(* PLC project SafeLOGIC, BrAutomation SafeDESIGNER  5.24.1.0 *)
(* stored: companyURL http://www.br-automation.com, creationDateTime Fri Nov 28 15:23:45 2025 *)

PROGRAM ERV_Fan

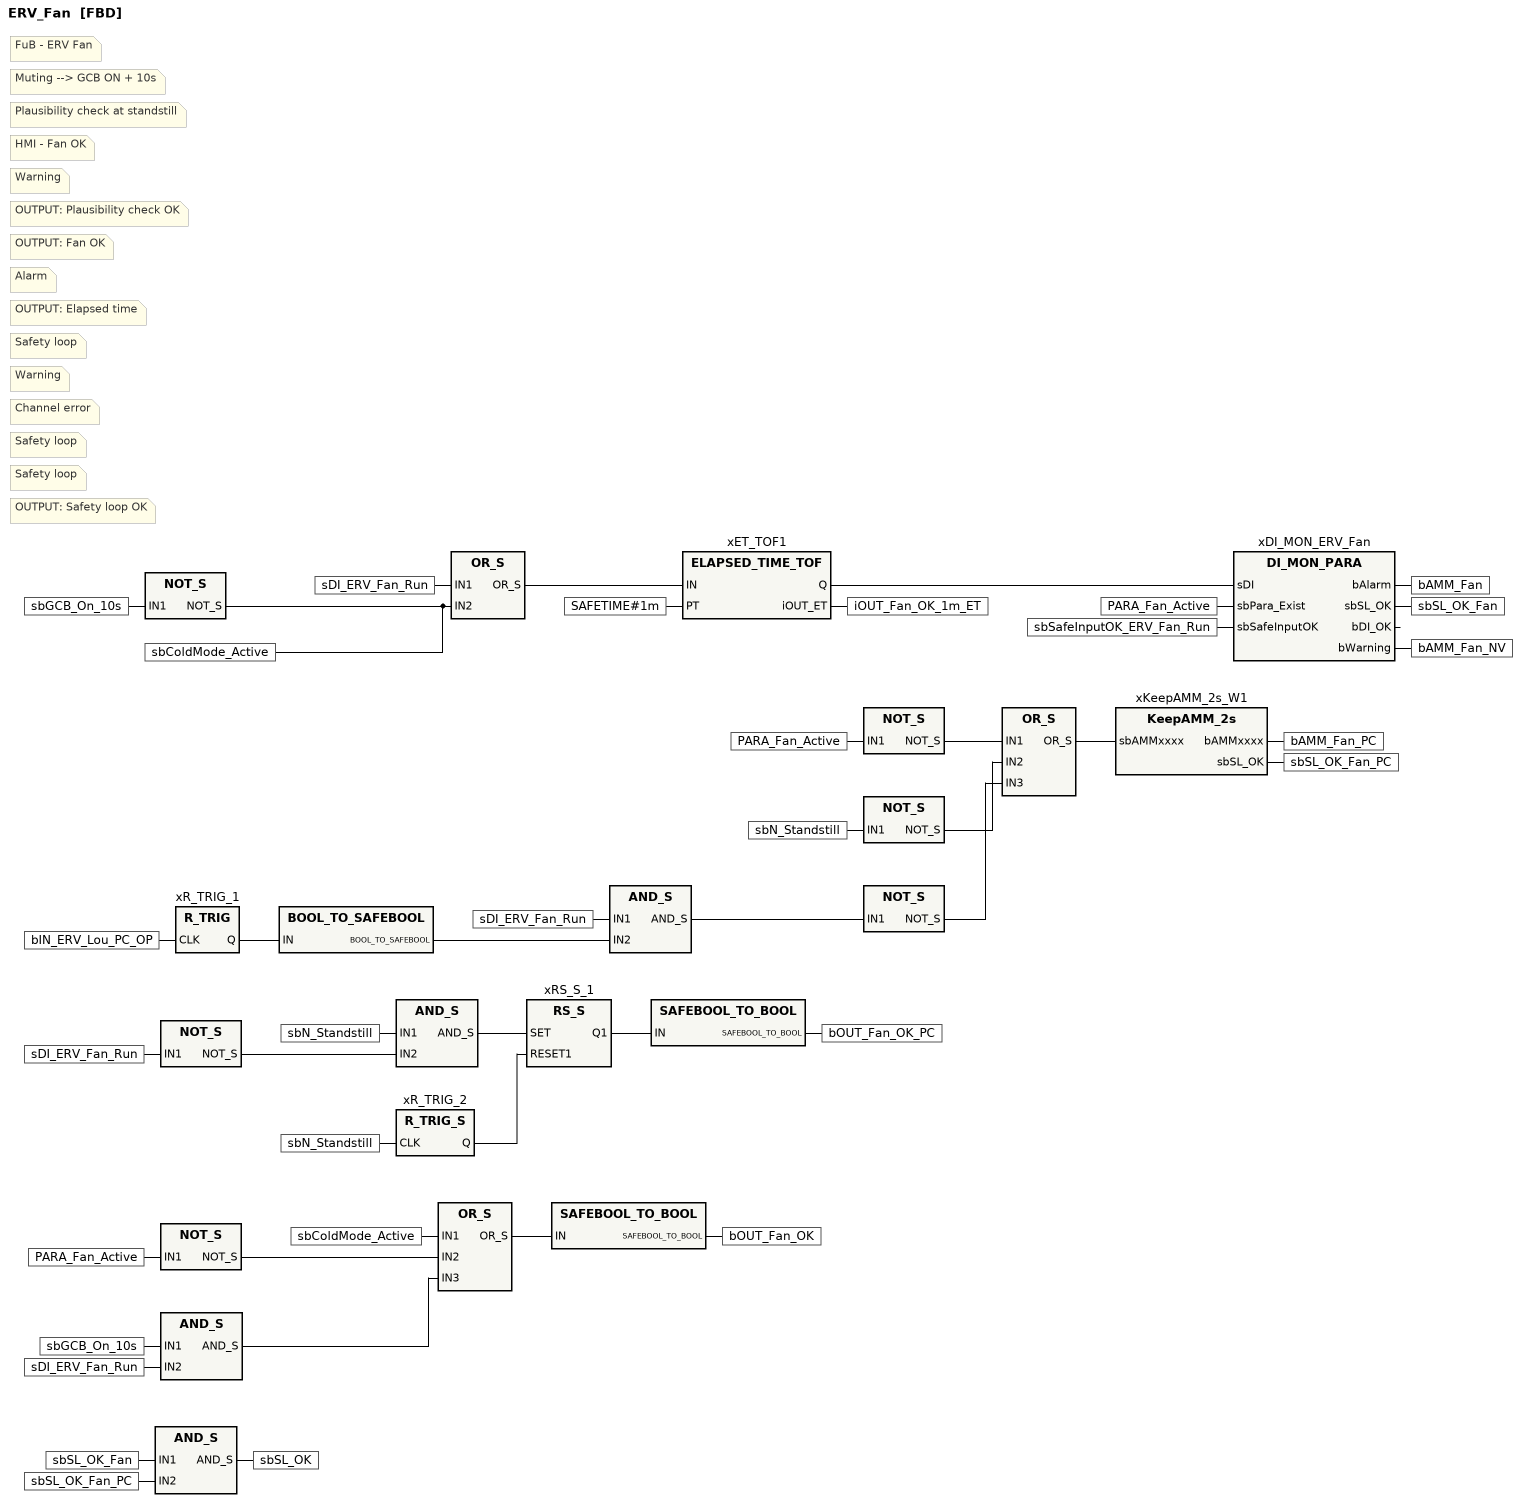
(* FBD diagram, written out as Structured Text *)
(* FuB - ERV Fan *)
(* Alarm *)
(* Safety loop *)
xET_TOF1(IN := OR_S(sDI_ERV_Fan_Run, sbColdMode_Active, NOT_S(sbGCB_On_10s)), PT := SAFETIME#1m);
xDI_MON_ERV_Fan(sDI := xET_TOF1.Q, sbPara_Exist := PARA_Fan_Active, sbSafeInputOK := sbSafeInputOK_ERV_Fan_Run);
bAMM_Fan := xDI_MON_ERV_Fan.bAlarm;
(* Muting --> GCB ON + 10s *)
(* Channel error *)
(* Warning *)
(* OUTPUT: Elapsed time *)
iOUT_Fan_OK_1m_ET := xET_TOF1.iOUT_ET;
bAMM_Fan_NV := xDI_MON_ERV_Fan.bWarning;
sbSL_OK_Fan := xDI_MON_ERV_Fan.sbSL_OK;
(* Plausibility check at standstill *)
(* Warning *)
(* Safety loop *)
xR_TRIG_1(CLK := bIN_ERV_Lou_PC_OP);
xKeepAMM_2s_W1(sbAMMxxxx := OR_S(NOT_S(PARA_Fan_Active), NOT_S(sbN_Standstill), NOT_S(AND_S(sDI_ERV_Fan_Run, BOOL_TO_SAFEBOOL(xR_TRIG_1.Q)))));
bAMM_Fan_PC := xKeepAMM_2s_W1.bAMMxxxx;
sbSL_OK_Fan_PC := xKeepAMM_2s_W1.sbSL_OK;
(* OUTPUT: Plausibility check OK *)
xR_TRIG_2(CLK := sbN_Standstill);
xRS_S_1(SET := AND_S(sbN_Standstill, NOT_S(sDI_ERV_Fan_Run)), RESET1 := xR_TRIG_2.Q);
bOUT_Fan_OK_PC := SAFEBOOL_TO_BOOL(xRS_S_1.Q1);
(* HMI - Fan OK *)
(* OUTPUT: Fan OK *)
bOUT_Fan_OK := SAFEBOOL_TO_BOOL(OR_S(sbColdMode_Active, NOT_S(PARA_Fan_Active), AND_S(sbGCB_On_10s, sDI_ERV_Fan_Run)));
(* Safety loop *)
(* OUTPUT: Safety loop OK *)
sbSL_OK := AND_S(sbSL_OK_Fan, sbSL_OK_Fan_PC);
END_PROGRAM
